FUNCTION_BLOCK MGE_HMI (* Service Interface Function Block Type *)
  (* Standard: 61499-2 *)
  (* Version 0.0, 17/03/2026, template *)
  PACKAGE Hidryco.HidrycoLib;
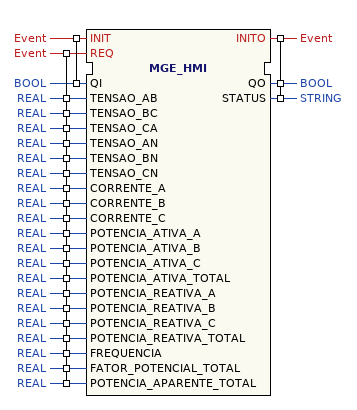
  EVENT_INPUT
    INIT WITH QI;
    REQ WITH TENSAO_AB, TENSAO_BC, TENSAO_CA, TENSAO_AN, TENSAO_BN, TENSAO_CN, CORRENTE_A, CORRENTE_B, CORRENTE_C, POTENCIA_ATIVA_A, POTENCIA_ATIVA_B, POTENCIA_ATIVA_C, POTENCIA_ATIVA_TOTAL, POTENCIA_REATIVA_A, POTENCIA_REATIVA_B, POTENCIA_REATIVA_C, POTENCIA_REATIVA_TOTAL, FREQUENCIA, FATOR_POTENCIAL_TOTAL, POTENCIA_APARENTE_TOTAL;
  END_EVENT
  EVENT_OUTPUT
    INITO WITH QO, STATUS;
  END_EVENT
  VAR_INPUT
    QI : BOOL;
    TENSAO_AB : REAL;
    TENSAO_BC : REAL;
    TENSAO_CA : REAL;
    TENSAO_AN : REAL;
    TENSAO_BN : REAL;
    TENSAO_CN : REAL;
    CORRENTE_A : REAL;
    CORRENTE_B : REAL;
    CORRENTE_C : REAL;
    POTENCIA_ATIVA_A : REAL;
    POTENCIA_ATIVA_B : REAL;
    POTENCIA_ATIVA_C : REAL;
    POTENCIA_ATIVA_TOTAL : REAL;
    POTENCIA_REATIVA_A : REAL;
    POTENCIA_REATIVA_B : REAL;
    POTENCIA_REATIVA_C : REAL;
    POTENCIA_REATIVA_TOTAL : REAL;
    FREQUENCIA : REAL;
    FATOR_POTENCIAL_TOTAL : REAL;
    POTENCIA_APARENTE_TOTAL : REAL;
  END_VAR
  VAR_OUTPUT
    QO : BOOL; (* Event Output Qualifier *)
    STATUS : STRING; (* Service Status *)
  END_VAR
  SERVICE /
    SEQUENCE 
    END_SEQUENCE
  END_SERVICE
END_FUNCTION_BLOCK
